// Mitsubishi GX Works2 project: PLC_GROUP15   PLC: FX3G

// global labels: Global1
VAR_GLOBAL
  StartDay AT X007 : BOOL;
  Input_Kadaif AT D1112 : REAL;
  Stock_Kadaif AT D1114 : REAL;
  Input_Pistachio AT D1108 : REAL;
  Input_Nuts AT D1104 : REAL;
  Stock_Nuts AT D1106 : REAL;
  Stock_Pistachio AT D1110 : REAL;
  Input_Chocolate AT D1100 : REAL;
  Stock_Chocolate AT D1102 : REAL;
  Srock_Filled AT M7 : BOOL;
  Stock_Filled AT M7 : BOOL;
END_VAR
VAR_GLOBAL CONSTANT
  Min_Pistachio : REAL := 120;
  Min_Kadaif : REAL := 60;
  Min_Nuts : REAL := 100;
  Min_Chocolate : REAL := 400;
END_VAR
VAR_GLOBAL
  Start_Day_Sign AT Y007 : BOOL;
  Start_Melt AT X001 : BOOL;
END_VAR
VAR_GLOBAL CONSTANT
  Reduce_Chocolate : REAL := 400;
END_VAR
VAR_GLOBAL
  Stock_MeltChocolate AT D1122 : REAL;
END_VAR
VAR_GLOBAL CONSTANT
  Add_Chocolate : REAL := 400;
END_VAR
VAR_GLOBAL
  Transferd AT M2 : BOOL;
  Melt_Time AT TC1 : BOOL;
  Degrees AT K30 : INT;
  Timers_Up AT TS1 : BOOL;
  Finish_Melt_Process AT M3 : BOOL;
  Melting_Lamp AT Y001 : BOOL;
  Place_Tavnit AT X003 : BOOL;
  Tavnit_Holder AT CC3 : BOOL;
  Four_Tavniut AT K4 : INT;
  Holder AT CS3 : BOOL;
END_VAR
VAR_GLOBAL CONSTANT
  Pour_Choclate : REAL := 400;
END_VAR
VAR_GLOBAL
  Chocolate_Poured AT M4 : BOOL;
  Casting_Time AT TC2 : BOOL;
  Seconds AT K40 : INT;
  Finish_Casting AT TS2 : BOOL;
  Finish_Timer AT TS2 : BOOL;
  Finished_Casting AT M5 : BOOL;
  Casting_Process AT Y002 : BOOL;
  Sample_From_Analog AT M4 : BOOL;
  Analog_Input AT D8281 : INT;
  Analog_Output AT D8282 : INT;
  Choose_Cream AT M6 : BOOL;
END_VAR
VAR_GLOBAL CONSTANT
  Min_Nuts_Cream : REAL;
  Max_Nuts_Cream : REAL := 2017;
  Min_Dubai_Cream : REAL := 2018;
  Max_Dubai_Cream : REAL := 4026;
  Nuts_Grams : REAL := 100;
  Pistachio_Grams : REAL := 100;
  NutsG : REAL := 20;
  PistachioG : REAL := 120;
  KadaifG : REAL := 60;
END_VAR
VAR_GLOBAL
  Dubai_Fill AT M10 : BOOL;
  Nuts_Fill AT M9 : BOOL;
  Glimmer_lights AT K50 : INT;
  Glimmer_Time AT TC4 : BOOL;
  Gliimer_Finished AT TS4 : BOOL;
  Glimmer_Stop AT M11 : BOOL;
  Glimerring AT M12 : BOOL;
  Glimmer_Second AT TC5 : BOOL;
  One_Second AT K10 : INT;
  Glimer_Seconds AT TS5 : BOOL;
  Another_Glimmer_Second AT TC6 : BOOL;
  Second_Light AT K10 : INT;
  Another_Glimmer_Seconds AT TS6 : BOOL;
  Second_Lights AT Y004 : BOOL;
  Kirur_Button AT X006 : BOOL;
  Kirur_Sec AT TC7 : BOOL;
  Kirur_Seconds AT K30 : INT;
  Kirur_Finished AT TS7 : BOOL;
  Kirur_Light AT Y006 : BOOL;
  Package AT X000 : BOOL;
  Ariza_Light AT Y005 : BOOL;
  Packaging AT CC5 : BOOL;
  Max_Packaging AT K4 : INT;
  Package_Finished AT CS5 : BOOL;
  Ariza_Storage AT D1116 : REAL;
END_VAR
VAR_GLOBAL CONSTANT
  Add_Ariza : REAL := 1;
END_VAR
VAR_GLOBAL
  Not_Enough_Materials AT M15 : BOOL;
END_VAR
VAR_GLOBAL CONSTANT
  Min_Kadaif1 : REAL := 60;
  Min_Pistachio1 : REAL := 120;
  Min_Nuts1 : REAL := 100;
  Min_Chocolate1 : REAL := 400;
END_VAR
VAR_GLOBAL
  Emergency_Button AT X005 : BOOL;
  Reset AT M16 : BOOL;
  Finish_Ariza AT M17 : BOOL;
END_VAR
VAR_GLOBAL CONSTANT
  Div_Analog1 : REAL := 40;
END_VAR
VAR_GLOBAL
  Num_Of_Arizot AT D1118 : REAL;
  Analog_Sample AT D1120 : REAL;
  Degree_Hayshan AT X002 : BOOL;
  Get_The_Sample_FromAnalog AT X004 : BOOL;
END_VAR
VAR_GLOBAL CONSTANT
  Div_Analog2 : INT;
END_VAR
VAR_GLOBAL
  Reset_Happened AT M55 : BOOL;
  ResetHelpers AT M50 : BOOL;
  First_Light AT Y003 : BOOL;
  Nuts_Cream_Choosed AT M21 : BOOL;
  Dubai_Cream_Choosed AT M8 : BOOL;
END_VAR

// task Task_01 (event TRUE, interval 0, priority 31): POU_01

PROGRAM POU_01
(* structured ladder/FBD written out as ST: instructions are called as NAME(EN, inputs, outputs); _pN, _eN, _tN stand for wires *)
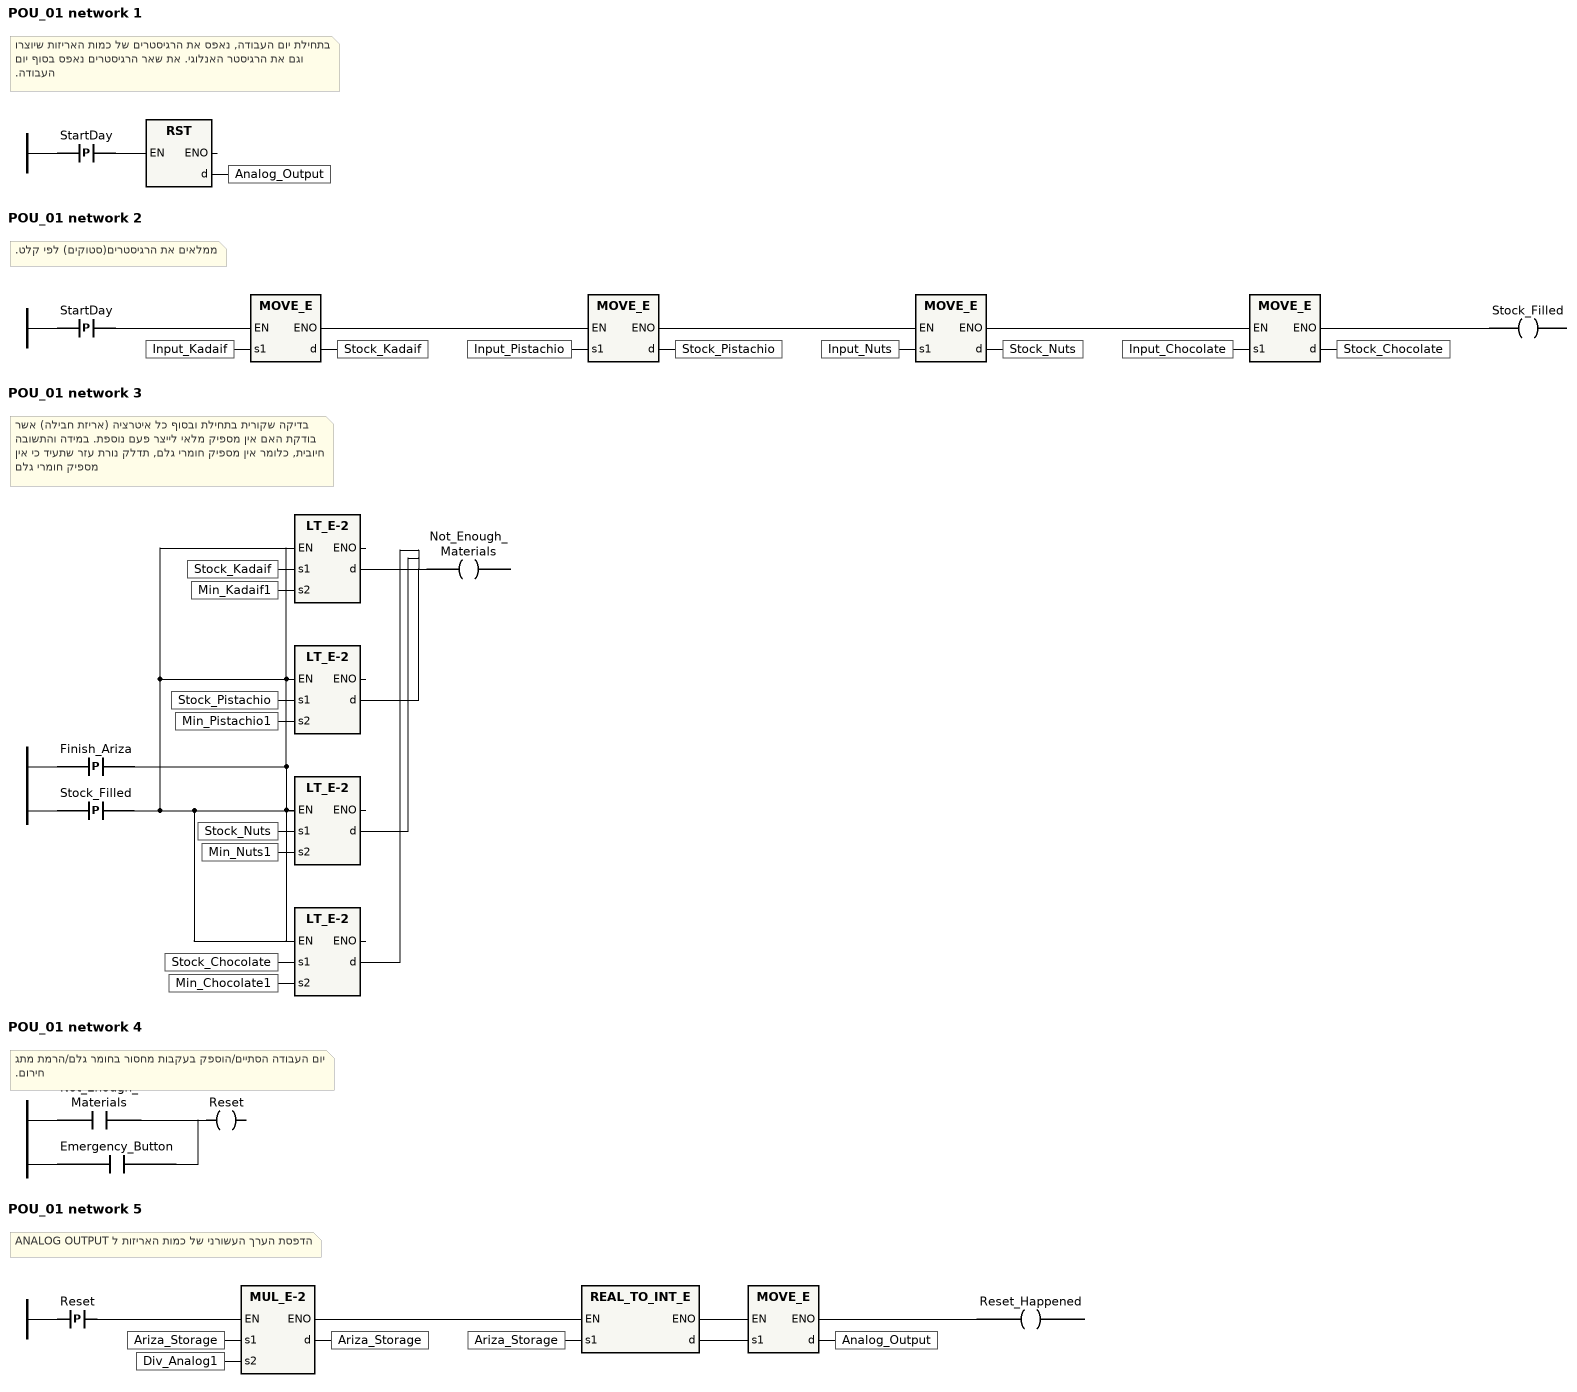
(* network 1 *)
(* בתחילת יום העבודה, נאפס את הרגיסטרים של כמות האריזות שיוצרו וגם את הרגיסטר האנלוגי. את שאר הרגיסטרים נאפס בסוף יום העבודה. *)
RST(LDP(TRUE, StartDay), Analog_Output);
(* network 2 *)
(* ממלאים את הרגיסטרים(סטוקים) לפי קלט. *)
_e1 := MOVE_E(LDP(TRUE, StartDay), Input_Kadaif, Stock_Kadaif);
_e2 := MOVE_E(_e1, Input_Pistachio, Stock_Pistachio);
_e3 := MOVE_E(_e2, Input_Nuts, Stock_Nuts);
_e4 := MOVE_E(_e3, Input_Chocolate, Stock_Chocolate);
Stock_Filled := _e4;
(* network 3 *)
(* בדיקה שקורית בתחילת ובסוף כל איטרציה (אריזת חבילה) אשר בודקת האם אין מספיק מלאי לייצר פעם נוספת. במידה והתשובה חיובית, כלומר אין מספיק חומרי גלם, תדלק נורת עזר שתעיד כי אין מספיק חומרי גלם *)
_p1 := LDP(TRUE, Finish_Ariza) OR LDP(TRUE, Stock_Filled);
LT_E(_p1, Stock_Kadaif, Min_Kadaif1, _t2);
LT_E(_p1, Stock_Pistachio, Min_Pistachio1, _t3);
LT_E(_p1, Stock_Nuts, Min_Nuts1, _t4);
LT_E(_p1, Stock_Chocolate, Min_Chocolate1, _t5);
Not_Enough_Materials := _t2 OR _t3 OR _t4 OR _t5;
(* network 4 *)
(* יום העבודה הסתיים/הוספק בעקבות מחסור בחומר גלם/הרמת מתג חירום. *)
Reset := Not_Enough_Materials OR Emergency_Button;
(* network 5 *)
(* הדפסת הערך העשורני של כמות האריזות ל ANALOG OUTPUT *)
_e1 := MUL_E(LDP(TRUE, Reset), Ariza_Storage, Div_Analog1, Ariza_Storage);
_e3 := REAL_TO_INT_E(_e1, Ariza_Storage, _t2);
_e4 := MOVE_E(_e3, _t2, Analog_Output);
Reset_Happened := _e4;
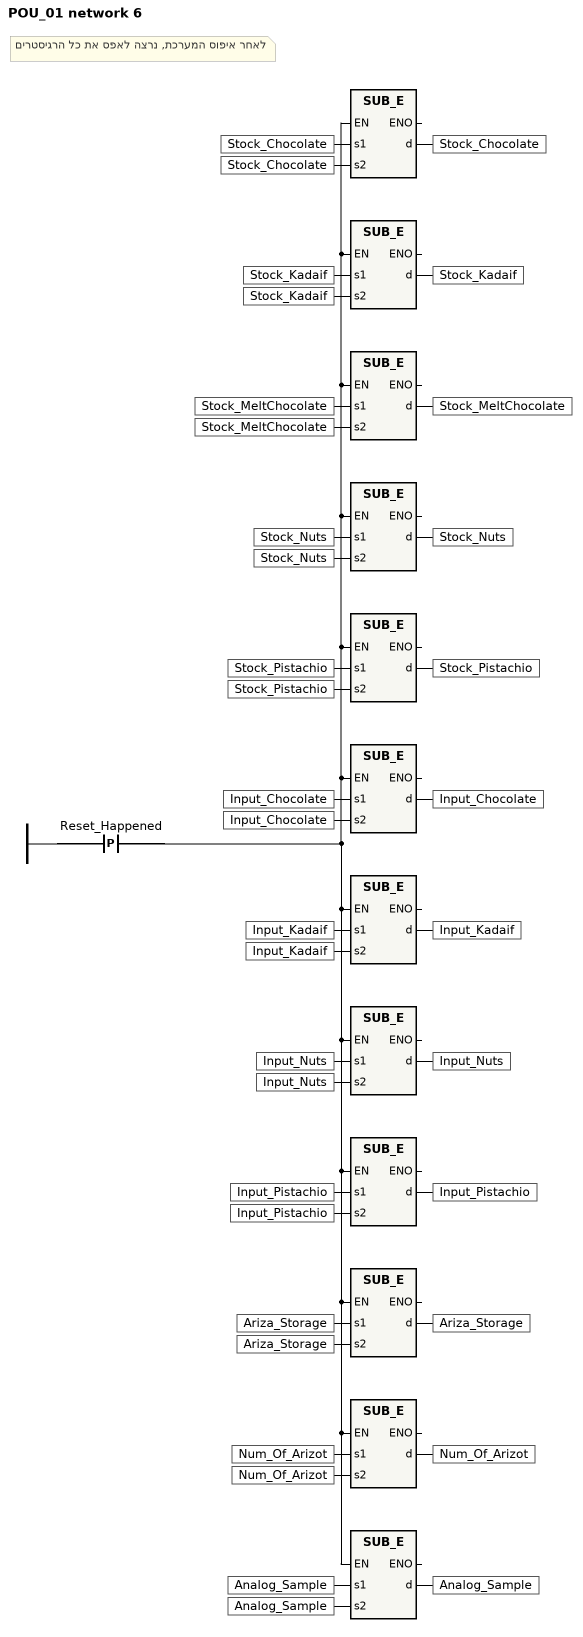
(* network 6 *)
(* לאחר איפוס המערכת, נרצה לאפס את כל הרגיסטרים *)
_p1 := LDP(TRUE, Reset_Happened);
SUB_E(_p1, Stock_Chocolate, Stock_Chocolate, Stock_Chocolate);
SUB_E(_p1, Stock_Kadaif, Stock_Kadaif, Stock_Kadaif);
SUB_E(_p1, Stock_MeltChocolate, Stock_MeltChocolate, Stock_MeltChocolate);
SUB_E(_p1, Stock_Nuts, Stock_Nuts, Stock_Nuts);
SUB_E(_p1, Stock_Pistachio, Stock_Pistachio, Stock_Pistachio);
SUB_E(_p1, Input_Chocolate, Input_Chocolate, Input_Chocolate);
SUB_E(_p1, Input_Kadaif, Input_Kadaif, Input_Kadaif);
SUB_E(_p1, Input_Nuts, Input_Nuts, Input_Nuts);
SUB_E(_p1, Input_Pistachio, Input_Pistachio, Input_Pistachio);
SUB_E(_p1, Ariza_Storage, Ariza_Storage, Ariza_Storage);
SUB_E(_p1, Num_Of_Arizot, Num_Of_Arizot, Num_Of_Arizot);
SUB_E(_p1, Analog_Sample, Analog_Sample, Analog_Sample);
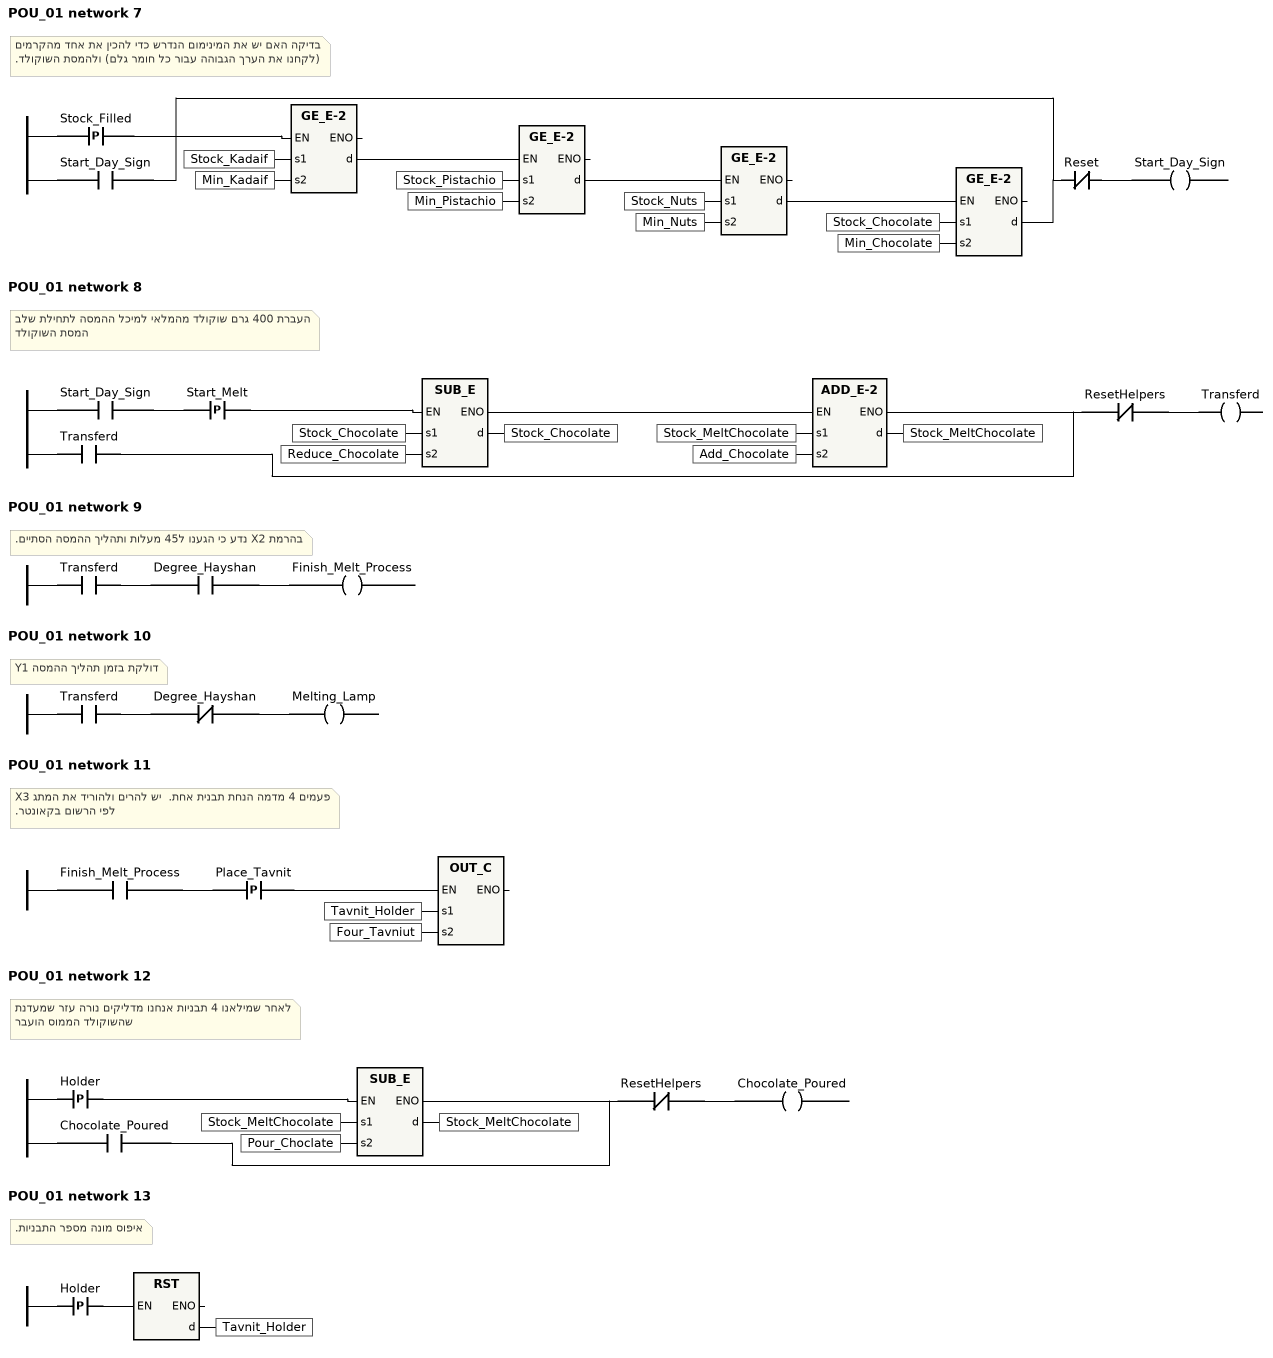
(* network 7 *)
(* בדיקה האם יש את המינימום הנדרש כדי להכין את אחד מהקרמים (לקחנו את הערך הגבוהה עבור כל חומר גלם) ולהמסת השוקולד. *)
GE_E(LDP(TRUE, Stock_Filled), Stock_Kadaif, Min_Kadaif, _t1);
GE_E(_t1, Stock_Pistachio, Min_Pistachio, _t2);
GE_E(_t2, Stock_Nuts, Min_Nuts, _t3);
GE_E(_t3, Stock_Chocolate, Min_Chocolate, _t4);
Start_Day_Sign := (_t4 OR Start_Day_Sign) AND NOT Reset;
(* network 8 *)
(* העברת 400 גרם שוקולד מהמלאי למיכל ההמסה לתחילת שלב המסת השוקולד *)
_e1 := SUB_E(Start_Day_Sign AND LDP(TRUE, Start_Melt), Stock_Chocolate, Reduce_Chocolate, Stock_Chocolate);
_e2 := ADD_E(_e1, Stock_MeltChocolate, Add_Chocolate, Stock_MeltChocolate);
Transferd := (_e2 OR Transferd) AND NOT ResetHelpers;
(* network 9 *)
(* בהרמת X2 נדע כי הגענו ל45 מעלות ותהליך ההמסה הסתיים. *)
Finish_Melt_Process := Transferd AND Degree_Hayshan;
(* network 10 *)
(* Y1 דולקת בזמן תהליך ההמסה *)
Melting_Lamp := Transferd AND NOT Degree_Hayshan;
(* network 11 *)
(* X3 מדמה הנחת תבנית אחת.  יש להרים ולהוריד את המתג 4 פעמים לפי הרשום בקאונטר. *)
OUT_C(Finish_Melt_Process AND LDP(TRUE, Place_Tavnit), Tavnit_Holder, Four_Tavniut);
(* network 12 *)
(* לאחר שמילאנו 4 תבניות אנחנו מדליקים נורה עזר שמעדנת שהשוקולד הממוס הועבר *)
_e1 := SUB_E(LDP(TRUE, Holder), Stock_MeltChocolate, Pour_Choclate, Stock_MeltChocolate);
Chocolate_Poured := (_e1 OR Chocolate_Poured) AND NOT ResetHelpers;
(* network 13 *)
(* איפוס מונה מספר התבניות. *)
RST(LDP(TRUE, Holder), Tavnit_Holder);
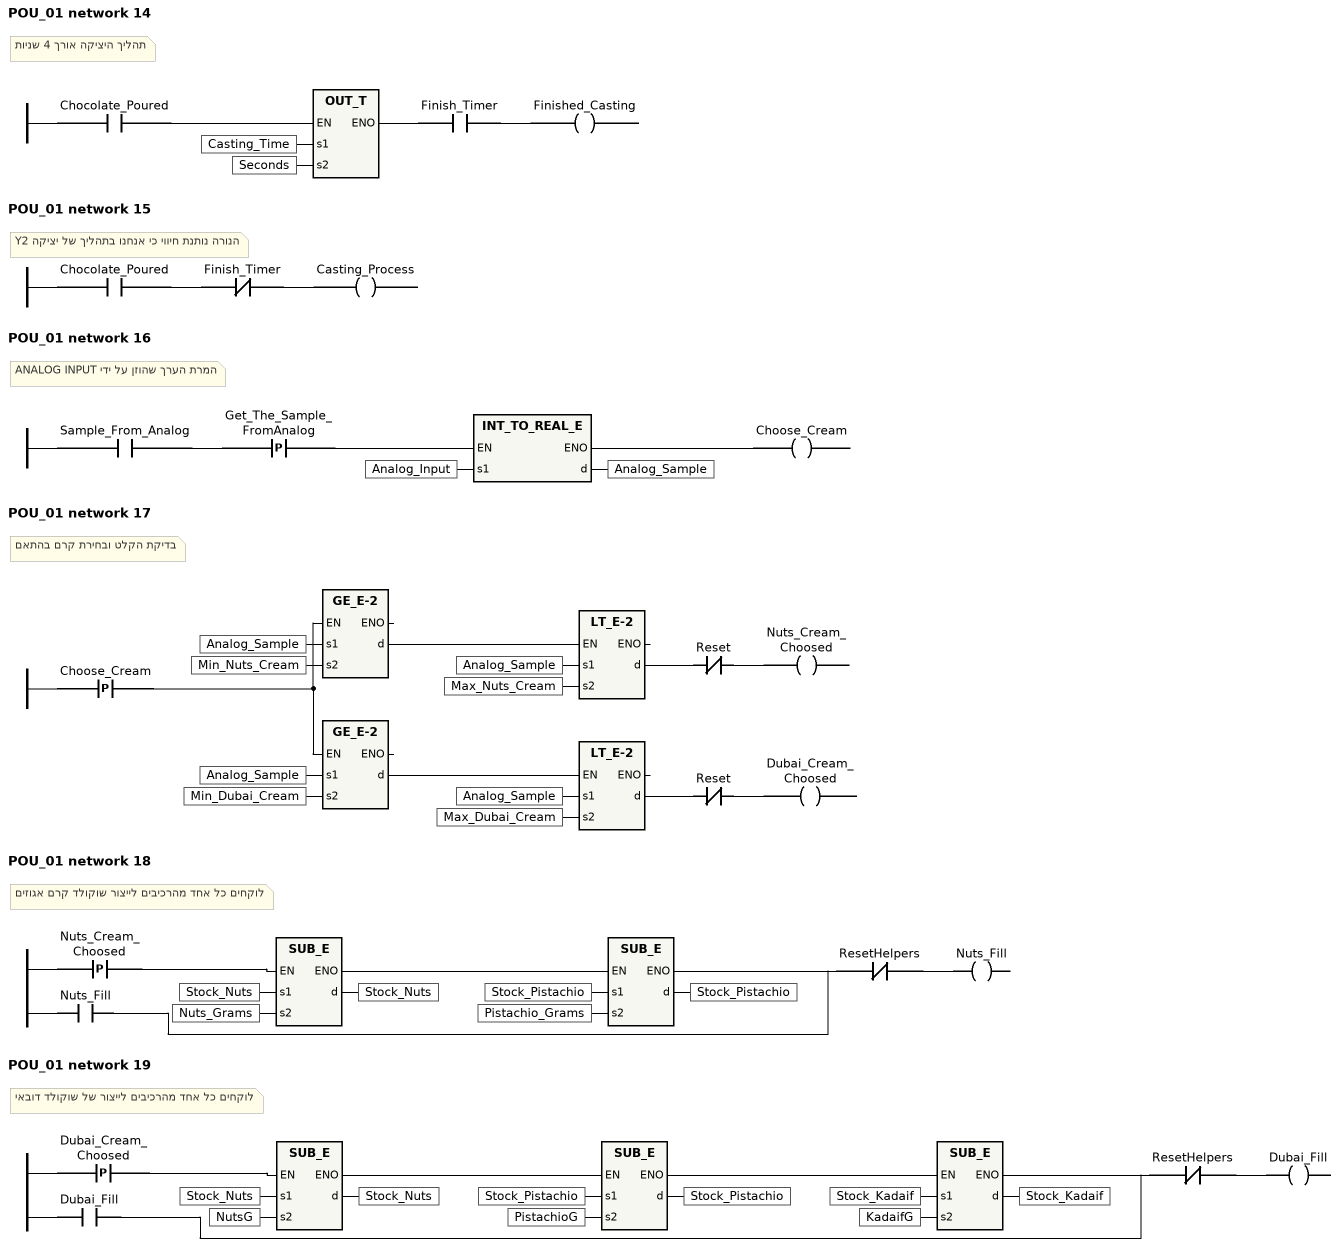
(* network 14 *)
(* תהליך היציקה אורך 4 שניות *)
_e1 := OUT_T(Chocolate_Poured, Casting_Time, Seconds);
Finished_Casting := _e1 AND Finish_Timer;
(* network 15 *)
(* הנורה נותנת חיווי כי אנחנו בתהליך של יציקה Y2 *)
Casting_Process := Chocolate_Poured AND NOT Finish_Timer;
(* network 16 *)
(* המרת הערך שהוזן על ידי ANALOG INPUT *)
_e1 := INT_TO_REAL_E(Sample_From_Analog AND LDP(TRUE, Get_The_Sample_FromAnalog), Analog_Input, Analog_Sample);
Choose_Cream := _e1;
(* network 17 *)
(* בדיקת הקלט ובחירת קרם בהתאם *)
_p1 := LDP(TRUE, Choose_Cream);
GE_E(_p1, Analog_Sample, Min_Nuts_Cream, _t2);
LT_E(_t2, Analog_Sample, Max_Nuts_Cream, _t3);
Nuts_Cream_Choosed := _t3 AND NOT Reset;
GE_E(_p1, Analog_Sample, Min_Dubai_Cream, _t4);
LT_E(_t4, Analog_Sample, Max_Dubai_Cream, _t5);
Dubai_Cream_Choosed := _t5 AND NOT Reset;
(* network 18 *)
(* לוקחים כל אחד מהרכיבים לייצור שוקולד קרם אגוזים *)
_e1 := SUB_E(LDP(TRUE, Nuts_Cream_Choosed), Stock_Nuts, Nuts_Grams, Stock_Nuts);
_e2 := SUB_E(_e1, Stock_Pistachio, Pistachio_Grams, Stock_Pistachio);
Nuts_Fill := (_e2 OR Nuts_Fill) AND NOT ResetHelpers;
(* network 19 *)
(* לוקחים כל אחד מהרכיבים לייצור של שוקולד דובאי *)
_e1 := SUB_E(LDP(TRUE, Dubai_Cream_Choosed), Stock_Nuts, NutsG, Stock_Nuts);
_e2 := SUB_E(_e1, Stock_Pistachio, PistachioG, Stock_Pistachio);
_e3 := SUB_E(_e2, Stock_Kadaif, KadaifG, Stock_Kadaif);
Dubai_Fill := (_e3 OR Dubai_Fill) AND NOT ResetHelpers;
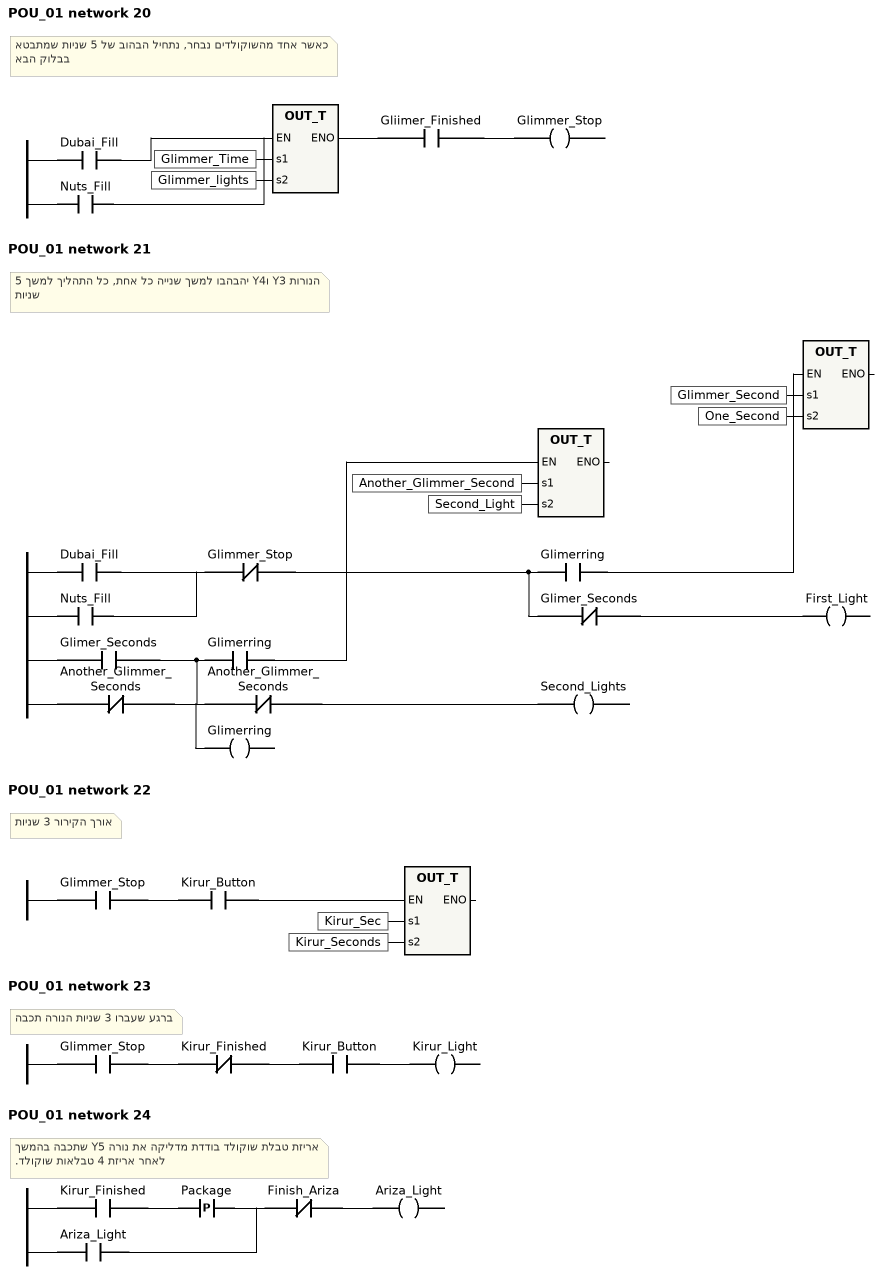
(* network 20 *)
(* כאשר אחד מהשוקולדים נבחר, נתחיל הבהוב של 5 שניות שמתבטא בבלוק הבא *)
_e1 := OUT_T(Dubai_Fill OR Nuts_Fill, Glimmer_Time, Glimmer_lights);
Glimmer_Stop := _e1 AND Gliimer_Finished;
(* network 21 *)
(* הנורות Y3 וY4 יהבהבו למשך שנייה כל אחת, כל התהליך למשך 5 שניות *)
_p1 := (Dubai_Fill OR Nuts_Fill) AND NOT Glimmer_Stop;
OUT_T(_p1 AND Glimerring, Glimmer_Second, One_Second);
First_Light := _p1 AND NOT Glimer_Seconds;
OUT_T(Glimer_Seconds AND Glimerring, Another_Glimmer_Second, Second_Light);
Second_Lights := Glimer_Seconds AND NOT Another_Glimmer_Seconds;
Glimerring := NOT Another_Glimmer_Seconds;
(* network 22 *)
(* אורך הקירור 3 שניות *)
OUT_T(Glimmer_Stop AND Kirur_Button, Kirur_Sec, Kirur_Seconds);
(* network 23 *)
(* ברגע שעברו 3 שניות הנורה תכבה *)
Kirur_Light := Glimmer_Stop AND NOT Kirur_Finished AND Kirur_Button;
(* network 24 *)
(* אריזת טבלת שוקולד בודדת מדליקה את נורה Y5 שתכבה בהמשך לאחר אריזת 4 טבלאות שוקולד. *)
Ariza_Light := ((Kirur_Finished AND LDP(TRUE, Package)) OR Ariza_Light) AND NOT Finish_Ariza;
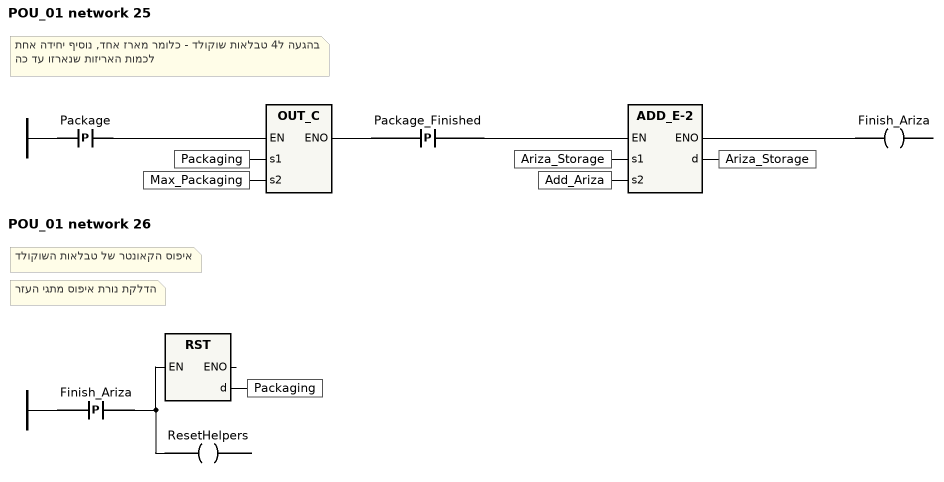
(* network 25 *)
(* בהגעה ל4 טבלאות שוקולד - כלומר מארז אחד, נוסיף יחידה אחת לכמות האריזות שנארזו עד כה *)
_e1 := OUT_C(LDP(TRUE, Package), Packaging, Max_Packaging);
_e2 := ADD_E(_e1 AND LDP(TRUE, Package_Finished), Ariza_Storage, Add_Ariza, Ariza_Storage);
Finish_Ariza := _e2;
(* network 26 *)
(* איפוס הקאונטר של טבלאות השוקולד *)
(* הדלקת נורת איפוס מתגי העזר *)
_p1 := LDP(TRUE, Finish_Ariza);
RST(_p1, Packaging);
ResetHelpers := _p1;
END_PROGRAM
